// TIA Portal V20 export
FUNCTION_BLOCK "CallSimulation"   // FB19, LAD
// stored: MemoryReserve 100, SetENOAutomatically false
   VAR
      instSimRotaryAxis { ExternalAccessible := 'False'; ExternalVisible := 'False'; ExternalWritable := 'False'} : Array[0..49] of "LER_SimHmiRotaryAxis";
      Unwindwe1 { S7_SetPoint := 'True'} : "LER_SimHmiRotaryAxis";
      IEC_Timer_0_Instance { S7_SetPoint := 'True'} : TON_TIME;
      "LER_SimAxis+_Axis07_pnp1X" { S7_SetPoint := 'True'} : "LER_SimAxis+";
      "LER_SimAxis+_Axis10_pnp1Z" { S7_SetPoint := 'True'} : "LER_SimAxis+";
      "LER_SimAxis+_Axis8_pnp2X" { S7_SetPoint := 'True'} : "LER_SimAxis+";
      "LER_SimAxis+_Axis13_pnp2Z" { S7_SetPoint := 'True'} : "LER_SimAxis+";
      "LER_SimAxis+_Axis12_pnp1Z" { S7_SetPoint := 'True'} : "LER_SimAxis+";
      "LER_SimAxis+_Axis14_pnp2Z" { S7_SetPoint := 'True'} : "LER_SimAxis+";
      "LER_SimAxis+_Axis34_cutterX" { S7_SetPoint := 'True'} : "LER_SimAxis+";
      "LER_SimAxis+_Axis35_cutterZ" { S7_SetPoint := 'True'} : "LER_SimAxis+";
      "LER_SimAxis-_Axis36_GripperX" { S7_SetPoint := 'True'} : "LER_SimAxis-";
      "LER_SimAxis+_Axis37_gripperZ" { S7_SetPoint := 'True'} : "LER_SimAxis+";
      "LER_SimAxis-_Axis32_StackTableZ" { S7_SetPoint := 'True'} : "LER_SimAxis-";
      "LER_SimAxis+_Axis21_roller" { S7_SetPoint := 'True'} : "LER_SimAxis+";
      "LER_SimAxis+_gripperAxis_C" { S7_SetPoint := 'True'} : "LER_SimAxis+";
      IEC_Timer_1_Instance { S7_SetPoint := 'True'} : TON_TIME;
      "LER_SimAxis+_Axis05_pnp1X" { S7_SetPoint := 'True'} : "LER_SimAxis+";
      "LER_SimAxis+_Axis06_pnp2X" { S7_SetPoint := 'True'} : "LER_SimAxis+";
   END_VAR
   VAR CONSTANT
      FALSE : Bool := FALSE;
      TRUE : Bool := TRUE;
   END_VAR
   VAR_TEMP   // added for the SCL form of the ladder/FBD networks
      _w1 : Bool;
      _w2 : Bool;
      _w3 : Bool;
      _w4 : Bool;
      _w5 : Bool;
      _w6 : Bool;
      _w7 : Bool;
      _w8 : Bool;
   END_VAR
BEGIN

REGION Network 1: SIMIT simulation currently running
   // The input "0.000CC1-KE50_I1.6_SimitRunning" is a life bit from SIMIT, which is always TRUE while SIMIT is running. The following actions are performed in that case:
   // - Simulation button in HMI is not shown when a SIMIT simulation is currently running
   // - Deactivate PLC internal simulation while SIMIT simulation is running
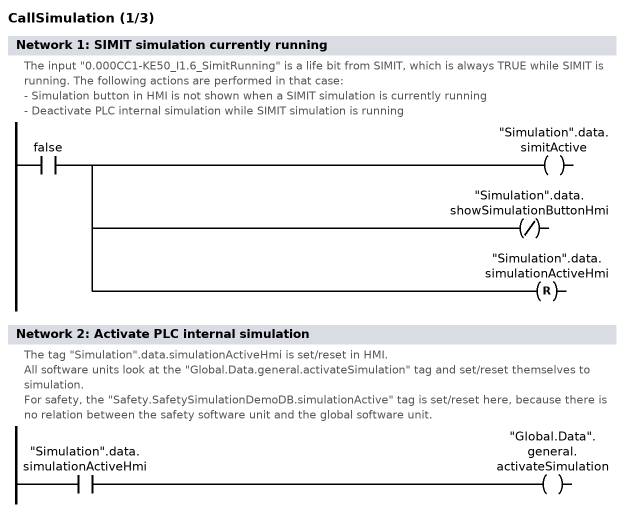
   RUNG wire#powerrail
      Contact( false )
      wire#w1
      Coil( "Simulation".data.simitActive )
   END_RUNG
   RUNG wire#w1
      I_Coil( "Simulation".data.showSimulationButtonHmi )
   END_RUNG
   RUNG wire#w1
      R_Coil( "Simulation".data.simulationActiveHmi )
   END_RUNG
   // the same network as SCL:
   "Simulation".data.simitActive := false;
   "Simulation".data.showSimulationButtonHmi := NOT false;
   IF false THEN "Simulation".data.simulationActiveHmi := FALSE; END_IF;
END_REGION

REGION Network 2: Activate PLC internal simulation
   // The tag "Simulation".data.simulationActiveHmi is set/reset in HMI.
   // 
   // All software units look at the "Global.Data.general.activateSimulation" tag and set/reset themselves to simulation.
   // 
   // For safety, the "Safety.SafetySimulationDemoDB.simulationActive" tag is set/reset here, because there is no relation between the safety software unit and the global software unit.
   RUNG wire#powerrail
      Contact( "Simulation".data.simulationActiveHmi )
      Coil( "Global.Data".general.activateSimulation )
   END_RUNG
   // the same network as SCL:
   "Global.Data".general.activateSimulation := "Simulation".data.simulationActiveHmi;
END_REGION

REGION Network 3: Simulation Linear Axis
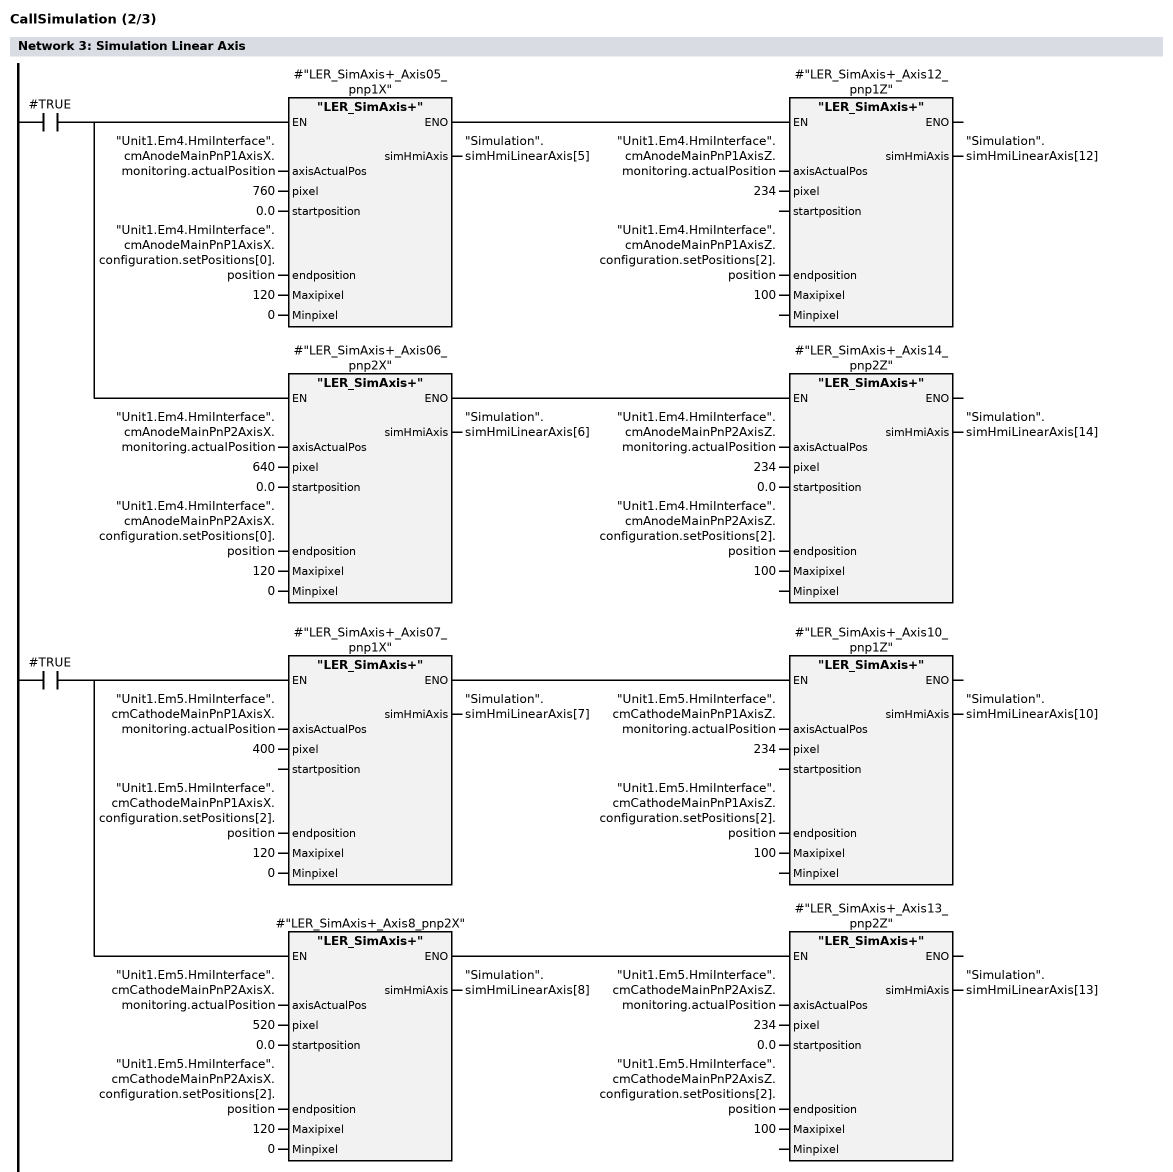
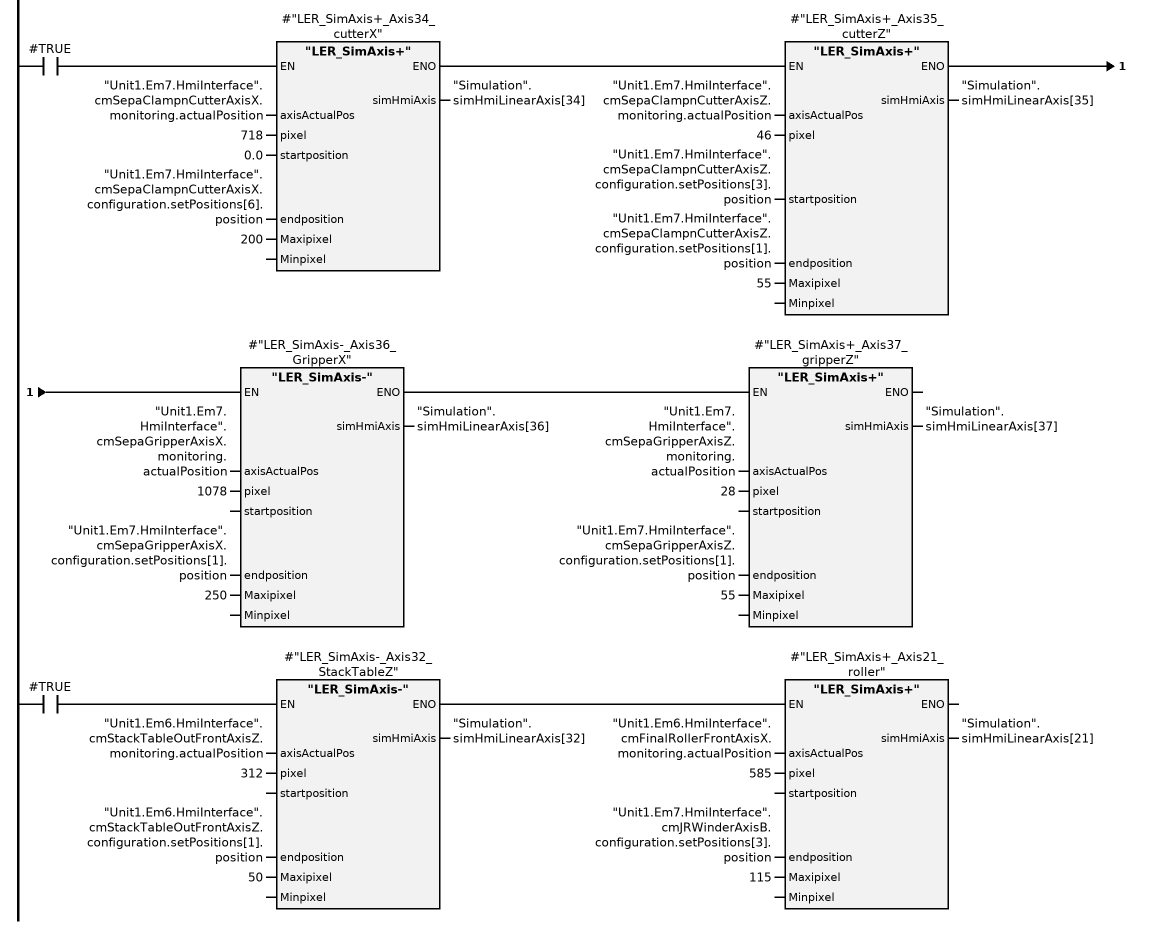
   RUNG wire#powerrail
      Contact( #TRUE )
      wire#w1
      #"LER_SimAxis+_Axis05_pnp1X"(axisActualPos := "Unit1.Em4.HmiInterface".cmAnodeMainPnP1AxisX.monitoring.actualPosition, pixel := 760, startposition := 0.0, endposition := "Unit1.Em4.HmiInterface".cmAnodeMainPnP1AxisX.configuration.setPositions[0].position, Maxipixel := 120, Minpixel := 0, simHmiAxis => "Simulation".simHmiLinearAxis[5])
      #"LER_SimAxis+_Axis12_pnp1Z"(axisActualPos := "Unit1.Em4.HmiInterface".cmAnodeMainPnP1AxisZ.monitoring.actualPosition, pixel := 234, startposition :=, endposition := "Unit1.Em4.HmiInterface".cmAnodeMainPnP1AxisZ.configuration.setPositions[2].position, Maxipixel := 100, Minpixel :=, simHmiAxis => "Simulation".simHmiLinearAxis[12])
   END_RUNG
   RUNG wire#w1
      #"LER_SimAxis+_Axis06_pnp2X"(axisActualPos := "Unit1.Em4.HmiInterface".cmAnodeMainPnP2AxisX.monitoring.actualPosition, pixel := 640, startposition := 0.0, endposition := "Unit1.Em4.HmiInterface".cmAnodeMainPnP2AxisX.configuration.setPositions[0].position, Maxipixel := 120, Minpixel := 0, simHmiAxis => "Simulation".simHmiLinearAxis[6])
      #"LER_SimAxis+_Axis14_pnp2Z"(axisActualPos := "Unit1.Em4.HmiInterface".cmAnodeMainPnP2AxisZ.monitoring.actualPosition, pixel := 234, startposition := 0.0, endposition := "Unit1.Em4.HmiInterface".cmAnodeMainPnP2AxisZ.configuration.setPositions[2].position, Maxipixel := 100, Minpixel :=, simHmiAxis => "Simulation".simHmiLinearAxis[14])
   END_RUNG
   RUNG wire#powerrail
      Contact( #TRUE )
      wire#w2
      #"LER_SimAxis+_Axis07_pnp1X"(axisActualPos := "Unit1.Em5.HmiInterface".cmCathodeMainPnP1AxisX.monitoring.actualPosition, pixel := 400, startposition :=, endposition := "Unit1.Em5.HmiInterface".cmCathodeMainPnP1AxisX.configuration.setPositions[2].position, Maxipixel := 120, Minpixel := 0, simHmiAxis => "Simulation".simHmiLinearAxis[7])
      #"LER_SimAxis+_Axis10_pnp1Z"(axisActualPos := "Unit1.Em5.HmiInterface".cmCathodeMainPnP1AxisZ.monitoring.actualPosition, pixel := 234, startposition :=, endposition := "Unit1.Em5.HmiInterface".cmCathodeMainPnP1AxisZ.configuration.setPositions[2].position, Maxipixel := 100, Minpixel :=, simHmiAxis => "Simulation".simHmiLinearAxis[10])
   END_RUNG
   RUNG wire#w2
      #"LER_SimAxis+_Axis8_pnp2X"(axisActualPos := "Unit1.Em5.HmiInterface".cmCathodeMainPnP2AxisX.monitoring.actualPosition, pixel := 520, startposition := 0.0, endposition := "Unit1.Em5.HmiInterface".cmCathodeMainPnP2AxisX.configuration.setPositions[2].position, Maxipixel := 120, Minpixel := 0, simHmiAxis => "Simulation".simHmiLinearAxis[8])
      #"LER_SimAxis+_Axis13_pnp2Z"(axisActualPos := "Unit1.Em5.HmiInterface".cmCathodeMainPnP2AxisZ.monitoring.actualPosition, pixel := 234, startposition := 0.0, endposition := "Unit1.Em5.HmiInterface".cmCathodeMainPnP2AxisZ.configuration.setPositions[2].position, Maxipixel := 100, Minpixel :=, simHmiAxis => "Simulation".simHmiLinearAxis[13])
   END_RUNG
   RUNG wire#powerrail
      Contact( #TRUE )
      #"LER_SimAxis+_Axis34_cutterX"(axisActualPos := "Unit1.Em7.HmiInterface".cmSepaClampnCutterAxisX.monitoring.actualPosition, pixel := 718, startposition := 0.0, endposition := "Unit1.Em7.HmiInterface".cmSepaClampnCutterAxisX.configuration.setPositions[6].position, Maxipixel := 200, Minpixel :=, simHmiAxis => "Simulation".simHmiLinearAxis[34])
      #"LER_SimAxis+_Axis35_cutterZ"(axisActualPos := "Unit1.Em7.HmiInterface".cmSepaClampnCutterAxisZ.monitoring.actualPosition, pixel := 46, startposition := "Unit1.Em7.HmiInterface".cmSepaClampnCutterAxisZ.configuration.setPositions[3].position, endposition := "Unit1.Em7.HmiInterface".cmSepaClampnCutterAxisZ.configuration.setPositions[1].position, Maxipixel := 55, Minpixel :=, simHmiAxis => "Simulation".simHmiLinearAxis[35])
      #"LER_SimAxis-_Axis36_GripperX"(axisActualPos := "Unit1.Em7.HmiInterface".cmSepaGripperAxisX.monitoring.actualPosition, pixel := 1078, startposition :=, endposition := "Unit1.Em7.HmiInterface".cmSepaGripperAxisX.configuration.setPositions[1].position, Maxipixel := 250, Minpixel :=, simHmiAxis => "Simulation".simHmiLinearAxis[36])
      #"LER_SimAxis+_Axis37_gripperZ"(axisActualPos := "Unit1.Em7.HmiInterface".cmSepaGripperAxisZ.monitoring.actualPosition, pixel := 28, startposition :=, endposition := "Unit1.Em7.HmiInterface".cmSepaGripperAxisZ.configuration.setPositions[1].position, Maxipixel := 55, Minpixel :=, simHmiAxis => "Simulation".simHmiLinearAxis[37])
   END_RUNG
   RUNG wire#powerrail
      Contact( #TRUE )
      #"LER_SimAxis-_Axis32_StackTableZ"(axisActualPos := "Unit1.Em6.HmiInterface".cmStackTableOutFrontAxisZ.monitoring.actualPosition, pixel := 312, startposition :=, endposition := "Unit1.Em6.HmiInterface".cmStackTableOutFrontAxisZ.configuration.setPositions[1].position, Maxipixel := 50, Minpixel :=, simHmiAxis => "Simulation".simHmiLinearAxis[32])
      #"LER_SimAxis+_Axis21_roller"(axisActualPos := "Unit1.Em6.HmiInterface".cmFinalRollerFrontAxisX.monitoring.actualPosition, pixel := 585, startposition :=, endposition := "Unit1.Em7.HmiInterface".cmJRWinderAxisB.configuration.setPositions[3].position, Maxipixel := 115, Minpixel :=, simHmiAxis => "Simulation".simHmiLinearAxis[21])
   END_RUNG
   // the same network as SCL:
   #"LER_SimAxis+_Axis05_pnp1X"(EN := #TRUE,   // "LER_SimAxis+"
                           axisActualPos := "Unit1.Em4.HmiInterface".cmAnodeMainPnP1AxisX.monitoring.actualPosition,
                           pixel := 760,
                           startposition := 0.0,
                           endposition := "Unit1.Em4.HmiInterface".cmAnodeMainPnP1AxisX.configuration.setPositions[0].position,
                           Maxipixel := 120,
                           Minpixel := 0,
                           simHmiAxis => "Simulation".simHmiLinearAxis[5],
                           ENO => #_w1);
   IF #_w1 THEN
       #"LER_SimAxis+_Axis12_pnp1Z"(axisActualPos := "Unit1.Em4.HmiInterface".cmAnodeMainPnP1AxisZ.monitoring.actualPosition,   // "LER_SimAxis+"
                               pixel := 234,
                               endposition := "Unit1.Em4.HmiInterface".cmAnodeMainPnP1AxisZ.configuration.setPositions[2].position,
                               Maxipixel := 100,
                               simHmiAxis => "Simulation".simHmiLinearAxis[12]);
   END_IF;
   #"LER_SimAxis+_Axis06_pnp2X"(EN := #TRUE,   // "LER_SimAxis+"
                           axisActualPos := "Unit1.Em4.HmiInterface".cmAnodeMainPnP2AxisX.monitoring.actualPosition,
                           pixel := 640,
                           startposition := 0.0,
                           endposition := "Unit1.Em4.HmiInterface".cmAnodeMainPnP2AxisX.configuration.setPositions[0].position,
                           Maxipixel := 120,
                           Minpixel := 0,
                           simHmiAxis => "Simulation".simHmiLinearAxis[6],
                           ENO => #_w2);
   IF #_w2 THEN
       #"LER_SimAxis+_Axis14_pnp2Z"(axisActualPos := "Unit1.Em4.HmiInterface".cmAnodeMainPnP2AxisZ.monitoring.actualPosition,   // "LER_SimAxis+"
                               pixel := 234,
                               startposition := 0.0,
                               endposition := "Unit1.Em4.HmiInterface".cmAnodeMainPnP2AxisZ.configuration.setPositions[2].position,
                               Maxipixel := 100,
                               simHmiAxis => "Simulation".simHmiLinearAxis[14]);
   END_IF;
   #"LER_SimAxis+_Axis07_pnp1X"(EN := #TRUE,   // "LER_SimAxis+"
                           axisActualPos := "Unit1.Em5.HmiInterface".cmCathodeMainPnP1AxisX.monitoring.actualPosition,
                           pixel := 400,
                           endposition := "Unit1.Em5.HmiInterface".cmCathodeMainPnP1AxisX.configuration.setPositions[2].position,
                           Maxipixel := 120,
                           Minpixel := 0,
                           simHmiAxis => "Simulation".simHmiLinearAxis[7],
                           ENO => #_w3);
   IF #_w3 THEN
       #"LER_SimAxis+_Axis10_pnp1Z"(axisActualPos := "Unit1.Em5.HmiInterface".cmCathodeMainPnP1AxisZ.monitoring.actualPosition,   // "LER_SimAxis+"
                               pixel := 234,
                               endposition := "Unit1.Em5.HmiInterface".cmCathodeMainPnP1AxisZ.configuration.setPositions[2].position,
                               Maxipixel := 100,
                               simHmiAxis => "Simulation".simHmiLinearAxis[10]);
   END_IF;
   #"LER_SimAxis+_Axis8_pnp2X"(EN := #TRUE,   // "LER_SimAxis+"
                           axisActualPos := "Unit1.Em5.HmiInterface".cmCathodeMainPnP2AxisX.monitoring.actualPosition,
                           pixel := 520,
                           startposition := 0.0,
                           endposition := "Unit1.Em5.HmiInterface".cmCathodeMainPnP2AxisX.configuration.setPositions[2].position,
                           Maxipixel := 120,
                           Minpixel := 0,
                           simHmiAxis => "Simulation".simHmiLinearAxis[8],
                           ENO => #_w4);
   IF #_w4 THEN
       #"LER_SimAxis+_Axis13_pnp2Z"(axisActualPos := "Unit1.Em5.HmiInterface".cmCathodeMainPnP2AxisZ.monitoring.actualPosition,   // "LER_SimAxis+"
                               pixel := 234,
                               startposition := 0.0,
                               endposition := "Unit1.Em5.HmiInterface".cmCathodeMainPnP2AxisZ.configuration.setPositions[2].position,
                               Maxipixel := 100,
                               simHmiAxis => "Simulation".simHmiLinearAxis[13]);
   END_IF;
   #"LER_SimAxis+_Axis34_cutterX"(EN := #TRUE,   // "LER_SimAxis+"
                           axisActualPos := "Unit1.Em7.HmiInterface".cmSepaClampnCutterAxisX.monitoring.actualPosition,
                           pixel := 718,
                           startposition := 0.0,
                           endposition := "Unit1.Em7.HmiInterface".cmSepaClampnCutterAxisX.configuration.setPositions[6].position,
                           Maxipixel := 200,
                           simHmiAxis => "Simulation".simHmiLinearAxis[34],
                           ENO => #_w5);
   #"LER_SimAxis+_Axis35_cutterZ"(EN := #_w5,   // "LER_SimAxis+"
                           axisActualPos := "Unit1.Em7.HmiInterface".cmSepaClampnCutterAxisZ.monitoring.actualPosition,
                           pixel := 46,
                           startposition := "Unit1.Em7.HmiInterface".cmSepaClampnCutterAxisZ.configuration.setPositions[3].position,
                           endposition := "Unit1.Em7.HmiInterface".cmSepaClampnCutterAxisZ.configuration.setPositions[1].position,
                           Maxipixel := 55,
                           simHmiAxis => "Simulation".simHmiLinearAxis[35],
                           ENO => #_w6);
   #"LER_SimAxis-_Axis36_GripperX"(EN := #_w6,   // "LER_SimAxis-"
                           axisActualPos := "Unit1.Em7.HmiInterface".cmSepaGripperAxisX.monitoring.actualPosition,
                           pixel := 1078,
                           endposition := "Unit1.Em7.HmiInterface".cmSepaGripperAxisX.configuration.setPositions[1].position,
                           Maxipixel := 250,
                           simHmiAxis => "Simulation".simHmiLinearAxis[36],
                           ENO => #_w7);
   IF #_w7 THEN
       #"LER_SimAxis+_Axis37_gripperZ"(axisActualPos := "Unit1.Em7.HmiInterface".cmSepaGripperAxisZ.monitoring.actualPosition,   // "LER_SimAxis+"
                               pixel := 28,
                               endposition := "Unit1.Em7.HmiInterface".cmSepaGripperAxisZ.configuration.setPositions[1].position,
                               Maxipixel := 55,
                               simHmiAxis => "Simulation".simHmiLinearAxis[37]);
   END_IF;
   #"LER_SimAxis-_Axis32_StackTableZ"(EN := #TRUE,   // "LER_SimAxis-"
                           axisActualPos := "Unit1.Em6.HmiInterface".cmStackTableOutFrontAxisZ.monitoring.actualPosition,
                           pixel := 312,
                           endposition := "Unit1.Em6.HmiInterface".cmStackTableOutFrontAxisZ.configuration.setPositions[1].position,
                           Maxipixel := 50,
                           simHmiAxis => "Simulation".simHmiLinearAxis[32],
                           ENO => #_w8);
   IF #_w8 THEN
       #"LER_SimAxis+_Axis21_roller"(axisActualPos := "Unit1.Em6.HmiInterface".cmFinalRollerFrontAxisX.monitoring.actualPosition,   // "LER_SimAxis+"
                               pixel := 585,
                               endposition := "Unit1.Em7.HmiInterface".cmJRWinderAxisB.configuration.setPositions[3].position,
                               Maxipixel := 115,
                               simHmiAxis => "Simulation".simHmiLinearAxis[21]);
   END_IF;
END_REGION

REGION Network 4: Simulation Rotary Axis
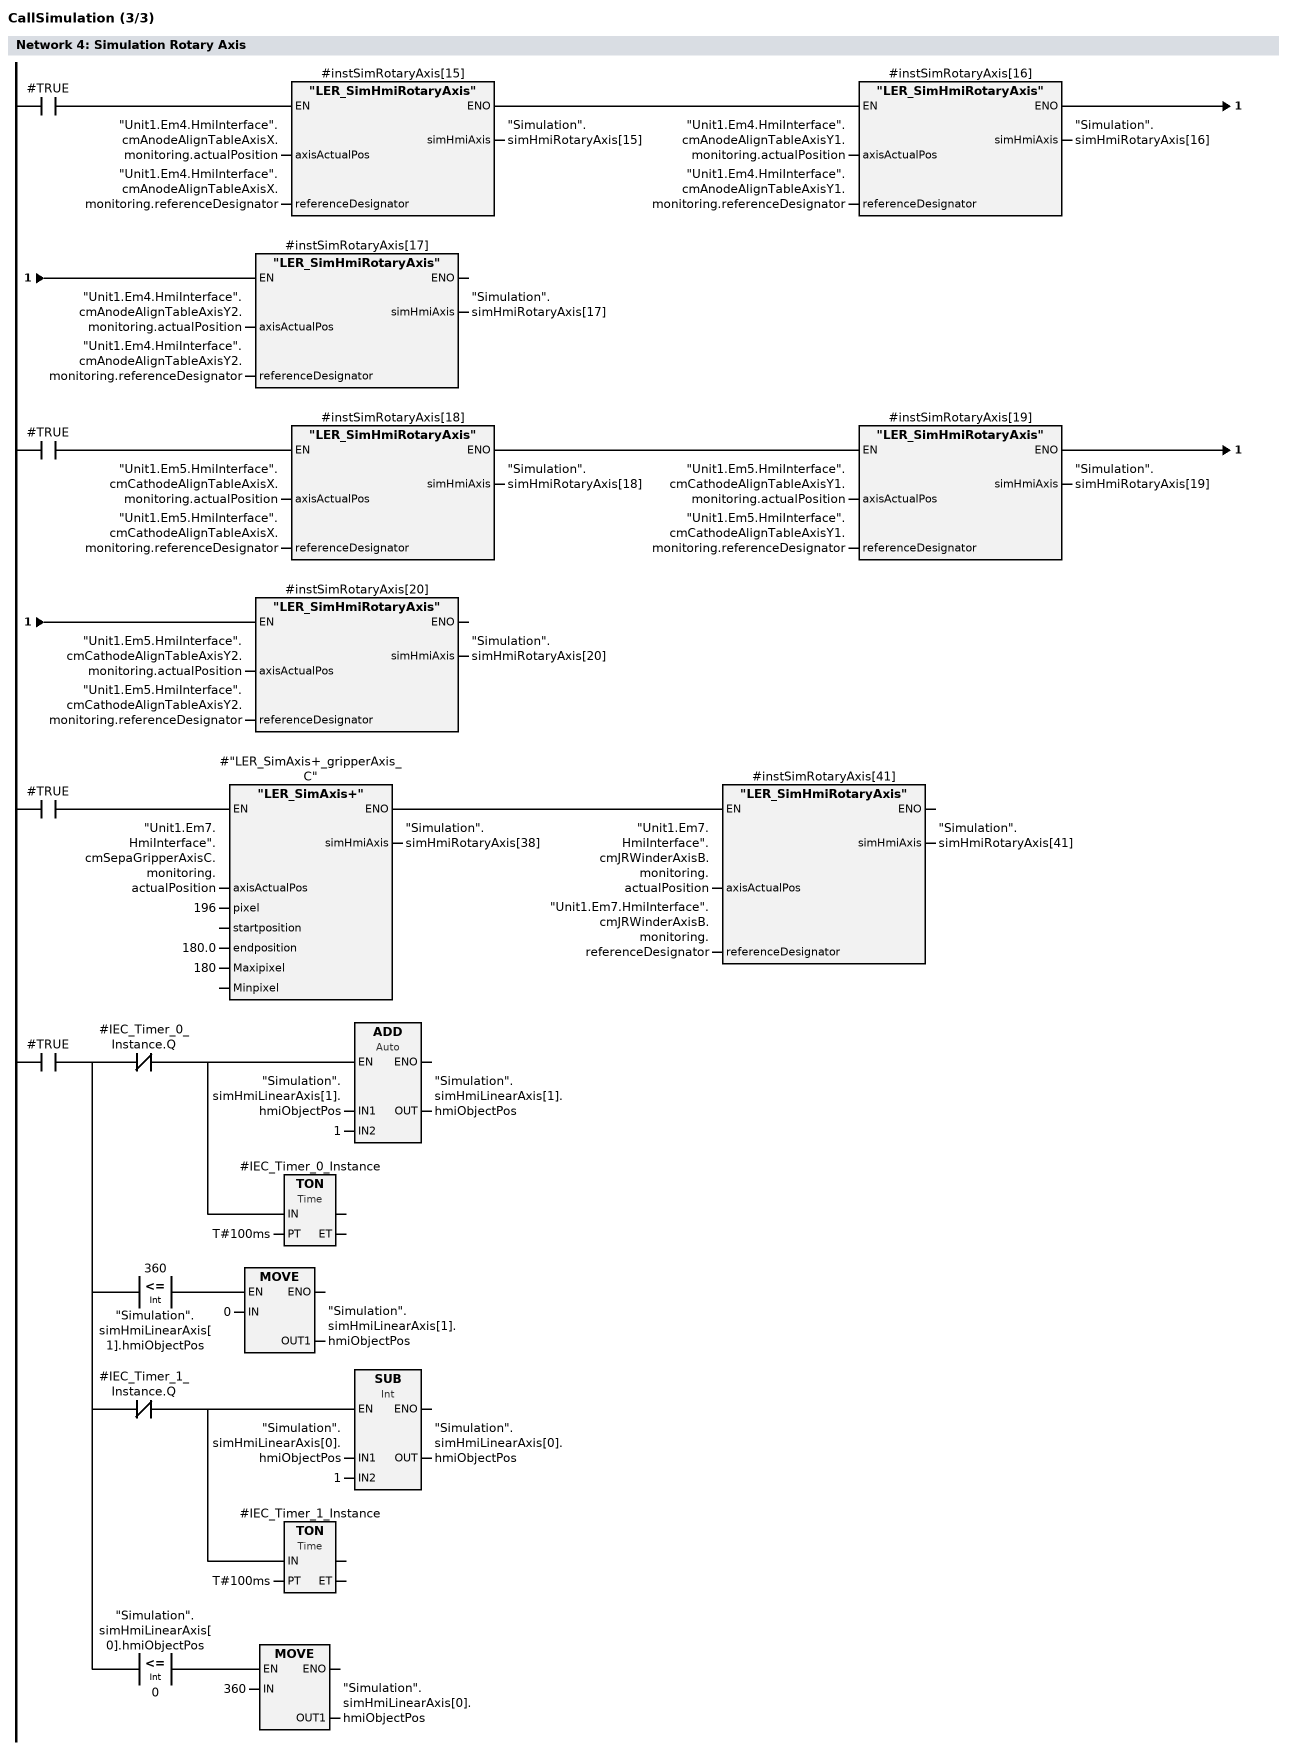
   RUNG wire#powerrail
      Contact( #TRUE )
      #instSimRotaryAxis[15](axisActualPos := "Unit1.Em4.HmiInterface".cmAnodeAlignTableAxisX.monitoring.actualPosition, referenceDesignator := "Unit1.Em4.HmiInterface".cmAnodeAlignTableAxisX.monitoring.referenceDesignator, simHmiAxis => "Simulation".simHmiRotaryAxis[15])
      #instSimRotaryAxis[16](axisActualPos := "Unit1.Em4.HmiInterface".cmAnodeAlignTableAxisY1.monitoring.actualPosition, referenceDesignator := "Unit1.Em4.HmiInterface".cmAnodeAlignTableAxisY1.monitoring.referenceDesignator, simHmiAxis => "Simulation".simHmiRotaryAxis[16])
      #instSimRotaryAxis[17](axisActualPos := "Unit1.Em4.HmiInterface".cmAnodeAlignTableAxisY2.monitoring.actualPosition, referenceDesignator := "Unit1.Em4.HmiInterface".cmAnodeAlignTableAxisY2.monitoring.referenceDesignator, simHmiAxis => "Simulation".simHmiRotaryAxis[17])
   END_RUNG
   RUNG wire#powerrail
      Contact( #TRUE )
      #instSimRotaryAxis[18](axisActualPos := "Unit1.Em5.HmiInterface".cmCathodeAlignTableAxisX.monitoring.actualPosition, referenceDesignator := "Unit1.Em5.HmiInterface".cmCathodeAlignTableAxisX.monitoring.referenceDesignator, simHmiAxis => "Simulation".simHmiRotaryAxis[18])
      #instSimRotaryAxis[19](axisActualPos := "Unit1.Em5.HmiInterface".cmCathodeAlignTableAxisY1.monitoring.actualPosition, referenceDesignator := "Unit1.Em5.HmiInterface".cmCathodeAlignTableAxisY1.monitoring.referenceDesignator, simHmiAxis => "Simulation".simHmiRotaryAxis[19])
      #instSimRotaryAxis[20](axisActualPos := "Unit1.Em5.HmiInterface".cmCathodeAlignTableAxisY2.monitoring.actualPosition, referenceDesignator := "Unit1.Em5.HmiInterface".cmCathodeAlignTableAxisY2.monitoring.referenceDesignator, simHmiAxis => "Simulation".simHmiRotaryAxis[20])
   END_RUNG
   RUNG wire#powerrail
      Contact( #TRUE )
      #"LER_SimAxis+_gripperAxis_C"(axisActualPos := "Unit1.Em7.HmiInterface".cmSepaGripperAxisC.monitoring.actualPosition, pixel := 196, startposition :=, endposition := 180.0, Maxipixel := 180, Minpixel :=, simHmiAxis => "Simulation".simHmiRotaryAxis[38])
      #instSimRotaryAxis[41](axisActualPos := "Unit1.Em7.HmiInterface".cmJRWinderAxisB.monitoring.actualPosition, referenceDesignator := "Unit1.Em7.HmiInterface".cmJRWinderAxisB.monitoring.referenceDesignator, simHmiAxis => "Simulation".simHmiRotaryAxis[41])
   END_RUNG
   RUNG wire#powerrail
      Contact( #TRUE )
      wire#w1
      I_Contact( #IEC_Timer_0_Instance.Q )
      wire#w2
      Add(in1 := "Simulation".simHmiLinearAxis[1].hmiObjectPos, in2 := 1, out => "Simulation".simHmiLinearAxis[1].hmiObjectPos)
   END_RUNG
   RUNG wire#w2
      { S7_Templates := "time_type := Time" } #IEC_Timer_0_Instance.TON(pt := T#100ms, et =>)
   END_RUNG
   RUNG wire#w1
      { S7_Templates := "SrcType := Int" } LE_Contact(in1 := 360, in2 := "Simulation".simHmiLinearAxis[1].hmiObjectPos)
      Move(in := 0, out1 => "Simulation".simHmiLinearAxis[1].hmiObjectPos)
   END_RUNG
   RUNG wire#w1
      I_Contact( #IEC_Timer_1_Instance.Q )
      wire#w3
      { S7_Templates := "SrcType := Int" } Sub(in1 := "Simulation".simHmiLinearAxis[0].hmiObjectPos, in2 := 1, out => "Simulation".simHmiLinearAxis[0].hmiObjectPos)
   END_RUNG
   RUNG wire#w3
      { S7_Templates := "time_type := Time" } #IEC_Timer_1_Instance.TON(pt := T#100ms, et =>)
   END_RUNG
   RUNG wire#w1
      { S7_Templates := "SrcType := Int" } LE_Contact(in1 := "Simulation".simHmiLinearAxis[0].hmiObjectPos, in2 := 0)
      Move(in := 360, out1 => "Simulation".simHmiLinearAxis[0].hmiObjectPos)
   END_RUNG
   // the same network as SCL:
   #instSimRotaryAxis[15](EN := #TRUE,   // "LER_SimHmiRotaryAxis"
                          axisActualPos := "Unit1.Em4.HmiInterface".cmAnodeAlignTableAxisX.monitoring.actualPosition,
                          referenceDesignator := "Unit1.Em4.HmiInterface".cmAnodeAlignTableAxisX.monitoring.referenceDesignator,
                          simHmiAxis => "Simulation".simHmiRotaryAxis[15],
                          ENO => #_w1);
   #instSimRotaryAxis[16](EN := #_w1,   // "LER_SimHmiRotaryAxis"
                          axisActualPos := "Unit1.Em4.HmiInterface".cmAnodeAlignTableAxisY1.monitoring.actualPosition,
                          referenceDesignator := "Unit1.Em4.HmiInterface".cmAnodeAlignTableAxisY1.monitoring.referenceDesignator,
                          simHmiAxis => "Simulation".simHmiRotaryAxis[16],
                          ENO => #_w2);
   IF #_w2 THEN
       #instSimRotaryAxis[17](axisActualPos := "Unit1.Em4.HmiInterface".cmAnodeAlignTableAxisY2.monitoring.actualPosition,   // "LER_SimHmiRotaryAxis"
                              referenceDesignator := "Unit1.Em4.HmiInterface".cmAnodeAlignTableAxisY2.monitoring.referenceDesignator,
                              simHmiAxis => "Simulation".simHmiRotaryAxis[17]);
   END_IF;
   #instSimRotaryAxis[18](EN := #TRUE,   // "LER_SimHmiRotaryAxis"
                          axisActualPos := "Unit1.Em5.HmiInterface".cmCathodeAlignTableAxisX.monitoring.actualPosition,
                          referenceDesignator := "Unit1.Em5.HmiInterface".cmCathodeAlignTableAxisX.monitoring.referenceDesignator,
                          simHmiAxis => "Simulation".simHmiRotaryAxis[18],
                          ENO => #_w3);
   #instSimRotaryAxis[19](EN := #_w3,   // "LER_SimHmiRotaryAxis"
                          axisActualPos := "Unit1.Em5.HmiInterface".cmCathodeAlignTableAxisY1.monitoring.actualPosition,
                          referenceDesignator := "Unit1.Em5.HmiInterface".cmCathodeAlignTableAxisY1.monitoring.referenceDesignator,
                          simHmiAxis => "Simulation".simHmiRotaryAxis[19],
                          ENO => #_w4);
   IF #_w4 THEN
       #instSimRotaryAxis[20](axisActualPos := "Unit1.Em5.HmiInterface".cmCathodeAlignTableAxisY2.monitoring.actualPosition,   // "LER_SimHmiRotaryAxis"
                              referenceDesignator := "Unit1.Em5.HmiInterface".cmCathodeAlignTableAxisY2.monitoring.referenceDesignator,
                              simHmiAxis => "Simulation".simHmiRotaryAxis[20]);
   END_IF;
   #"LER_SimAxis+_gripperAxis_C"(EN := #TRUE,   // "LER_SimAxis+"
                           axisActualPos := "Unit1.Em7.HmiInterface".cmSepaGripperAxisC.monitoring.actualPosition,
                           pixel := 196,
                           endposition := 180.0,
                           Maxipixel := 180,
                           simHmiAxis => "Simulation".simHmiRotaryAxis[38],
                           ENO => #_w5);
   IF #_w5 THEN
       #instSimRotaryAxis[41](axisActualPos := "Unit1.Em7.HmiInterface".cmJRWinderAxisB.monitoring.actualPosition,   // "LER_SimHmiRotaryAxis"
                              referenceDesignator := "Unit1.Em7.HmiInterface".cmJRWinderAxisB.monitoring.referenceDesignator,
                              simHmiAxis => "Simulation".simHmiRotaryAxis[41]);
   END_IF;
   #_w6 := #TRUE AND NOT #IEC_Timer_0_Instance.Q;
   IF #_w6 THEN
       "Simulation".simHmiLinearAxis[1].hmiObjectPos := "Simulation".simHmiLinearAxis[1].hmiObjectPos + 1;
   END_IF;
   #IEC_Timer_0_Instance(IN := #_w6, PT := T#100ms);   // TON
   IF #TRUE AND (360 <= "Simulation".simHmiLinearAxis[1].hmiObjectPos) THEN
       "Simulation".simHmiLinearAxis[1].hmiObjectPos := 0;
   END_IF;
   #_w7 := #TRUE AND NOT #IEC_Timer_1_Instance.Q;
   IF #_w7 THEN
       "Simulation".simHmiLinearAxis[0].hmiObjectPos := "Simulation".simHmiLinearAxis[0].hmiObjectPos - 1;
   END_IF;
   #IEC_Timer_1_Instance(IN := #_w7, PT := T#100ms);   // TON
   IF #TRUE AND ("Simulation".simHmiLinearAxis[0].hmiObjectPos <= 0) THEN
       "Simulation".simHmiLinearAxis[0].hmiObjectPos := 360;
   END_IF;
END_REGION
END_FUNCTION_BLOCK
